// TwinCAT 3 PLC project PupunPLC
// ProgramVersion: 3.1.4024.0
// libraries:
//   Tc2_Standard, * (Beckhoff Automation GmbH)
//   Tc2_System, * (Beckhoff Automation GmbH)
//   Tc3_Module, * (Beckhoff Automation GmbH)
// project tree:
//   FactoryIO/GVLs/ GVL_Tutti.TcGVL
//   FactoryIO/TUTTITEHDAS/01 IN AND SORT/ FB_PICKNPLACE.TcPOU, FB_SPECIAL.TcPOU, FB_TURNTABLE.TcPOU, FB_WEIGHT.TcPOU
//   FactoryIO/TUTTITEHDAS/02 CNC/ FB_CNC_MILL.TcPOU, FB_WHEELSORT.TcPOU
//   FactoryIO/TUTTITEHDAS/03 BOXING/ FB_CLAMP.TcPOU, FB_SPECIAL_2.TcPOU, FB_TWO_AXIS_PICK.TcPOU
//   FactoryIO/TUTTITEHDAS/04 STORAGE/ FB_STACKER.TcPOU
//   FactoryIO/TUTTITEHDAS/CONVEYORS/ FB_CONVEYOR1.TcPOU
//   FactoryIO/TUTTITEHDAS/DUT/ S_NAMES_IN.TcDUT, S_NAMES_OUT.TcDUT, S_REGS_IN.TcDUT, S_REGS_OUT.TcDUT, U_TRANSLATE_IN.TcDUT, U_TRANSLATE_OUT.TcDUT, U_TRANSLATE_REGS_IN.TcDUT, U_TRANSLATE_REGS_OUT.TcDUT
//   FactoryIO/TUTTITEHDAS/ FBD_TUTTILINJASTO.TcPOU, MAIN_TUTTI.TcPOU, RUN.TcPOU
//   FactoryIO/TUTTITEHDAS/GVL/ TIO.TcGVL
//   GVLs/ GVL.TcGVL
//   / PlcTask.TcTTO
//   POUs/ MAIN.TcPOU
// real-time tasks:
//   TASK PlcTask: cycle T#10ms, priority 20, ADS port 350

CONFIGURATION PupunPLC
    RESOURCE PLC ON TwinCAT3
        TASK PlcTask(INTERVAL := T#10ms, PRIORITY := 20);
        PROGRAM MAIN WITH PlcTask : MAIN;
    END_RESOURCE
END_CONFIGURATION

// ---- FactoryIO/TUTTITEHDAS/DUT/S_NAMES_IN.TcDUT
TYPE S_NAMES_IN :
STRUCT
			
//===== 	BYTE	0		
iInput0		:		BIT;
iInput1		:		BIT;
iInput2		:		BIT;
iInput3		:		BIT;
iInput4		:		BIT;
iInput5		:		BIT;
iSensor6	:		BIT;
iInput7		:		BIT;
//===== 	BYTE	1	
iInput8		:		BIT;
iInput9		:		BIT;
iInput10	:		BIT;
iInput11	:		BIT;
iInput12	:		BIT;
iRetroSensor1	:		BIT;
iRetroSensor2	:		BIT;
iInput15	:		BIT;
//===== 	BYTE	2	
iSortLimit0	:		BIT;
iSortLimit90:		BIT;
iSortBackLimit	:		BIT;
iSortFrontLimit	:		BIT;
iPickPlace_Climit:		BIT;
iPickPlace_Z_Moving	:		BIT;
iPickPlace_XY_Moving	:		BIT;
iPickPlace_BoxDetected	:		BIT;
//===== 	BYTE	3	
iInput24	:		BIT;
iInput25	:		BIT;
iInput26	:		BIT;
iInput27	:		BIT;
iInput28	:		BIT;
iInput29	:		BIT;
iPusherBackLimit	:		BIT;
iPusherFrontLimit	:		BIT;
//===== 	BYTE	4	
iInput32	:		BIT;
iInput33	:		BIT;
iInput34	:		BIT;
iSensor5	:		BIT;
iInput36	:		BIT;
iInput37	:		BIT;
iInput38	:		BIT;
iInput39	:		BIT;
//===== 	BYTE	5	
iCNC1_Opened	:		BIT;
iCNC1_Busy	:		BIT;
iCNC1_Error	:		BIT;
iCNC2_Opened	:		BIT;
iCNC2_Busy	:		BIT;
iCNC2_Error	:		BIT;
iCNC3_Opened	:		BIT;
iCNC3_Busy	:		BIT;
//===== 	BYTE	6	
iCNC3_Error	:		BIT;
iInput49	:		BIT;
iInput50	:		BIT;
iInput51	:		BIT;
iInput52	:		BIT;
iInput53	:		BIT;
iTwoAxisPick1_ItemDetected	:		BIT;
iSensor10	:		BIT;
//===== 	BYTE	7	
iClamp1_Limit	:		BIT;
iClamp1_Clamped	:		BIT;
iInput58	:		BIT;
iInput59	:		BIT;
iInput60	:		BIT;
iInput61	:		BIT;
Sensor11	:		BIT;
Stacker1_LeftLimit	:		BIT;
//===== 	BYTE	8	
Stacker1_RightLimit	:		BIT;
Stacker1_MiddleLimit:		BIT;
iInput66	:		BIT;
iInput67	:		BIT;
iInput68	:		BIT;
iInput69	:		BIT;
iInput70	:		BIT;
iInput71	:		BIT;
//===== 	BYTE	9	
iInput72	:		BIT;
iInput73	:		BIT;
iInput74	:		BIT;
iInput75	:		BIT;
iInput76	:		BIT;
iInput77	:		BIT;
iInput78	:		BIT;
iInput79	:		BIT;
//===== 	BYTE	10	
iInput80	:		BIT;
iInput81	:		BIT;
iInput82	:		BIT;
iInput83	:		BIT;
iInput84	:		BIT;
iInput85	:		BIT;
iInput86	:		BIT;
iInput87	:		BIT;
//===== 	BYTE	11	
iInput88	:		BIT;
iInput89	:		BIT;
iInput90	:		BIT;
iInput91	:		BIT;
iInput92	:		BIT;
iInput93	:		BIT;
iInput94	:		BIT;
iInput95	:		BIT;
//===== 	BYTE	12	
iInput96	:		BIT;
iInput97	:		BIT;
iInput98	:		BIT;
iInput99	:		BIT;
iInput100	:		BIT;
iInput101	:		BIT;
iInput102	:		BIT;
iInput103	:		BIT;
//===== 	BYTE	13	
iInput104	:		BIT;
iInput105	:		BIT;
iInput106	:		BIT;
iInput107	:		BIT;
iInput108	:		BIT;
iInput109	:		BIT;
iInput110	:		BIT;
iInput111	:		BIT;
//===== 	BYTE	14	
iInput112	:		BIT;
iInput113	:		BIT;
iInput114	:		BIT;
iInput115	:		BIT;
iInput116	:		BIT;
iInput117	:		BIT;
iInput118	:		BIT;
iInput119	:		BIT;
//===== 	BYTE	15	
iInput120	:		BIT;
iInput121	:		BIT;
iInput122	:		BIT;
iInput123	:		BIT;
iInput124	:		BIT;
iInput125	:		BIT;
iInput126	:		BIT;
iInput127	:		BIT;
//===== 	BYTE	16	
iInput128	:		BIT;
iInput129	:		BIT;
iInput130	:		BIT;
iInput131	:		BIT;
iInput132	:		BIT;
iInput133	:		BIT;
iInput134	:		BIT;
iInput135	:		BIT;
//===== 	BYTE	17	
iInput136	:		BIT;
iInput137	:		BIT;
iInput138	:		BIT;
iInput139	:		BIT;
iInput140	:		BIT;
iInput141	:		BIT;
iInput142	:		BIT;
iInput143	:		BIT;
//===== 	BYTE	18	
iInput144	:		BIT;
iInput145	:		BIT;
iInput146	:		BIT;
iInput147	:		BIT;
iInput148	:		BIT;
iInput149	:		BIT;
iInput150	:		BIT;
iInput151	:		BIT;
//===== 	BYTE	19	
iInput152	:		BIT;
iInput153	:		BIT;
iInput154	:		BIT;
iInput155	:		BIT;
iInput156	:		BIT;
iInput157	:		BIT;
iInput158	:		BIT;
iInput159	:		BIT;
//===== 	BYTE	20	
iInput160	:		BIT;
iInput161	:		BIT;
iInput162	:		BIT;
iInput163	:		BIT;
iInput164	:		BIT;
iInput165	:		BIT;
iInput166	:		BIT;
iInput167	:		BIT;
//===== 	BYTE	21	
iInput168	:		BIT;
iInput169	:		BIT;
iInput170	:		BIT;
iInput171	:		BIT;
iInput172	:		BIT;
iInput173	:		BIT;
iInput174	:		BIT;
iInput175	:		BIT;
//===== 	BYTE	22	
iInput176	:		BIT;
iInput177	:		BIT;
iInput178	:		BIT;
iInput179	:		BIT;
iInput180	:		BIT;
iInput181	:		BIT;
iInput182	:		BIT;
iInput183	:		BIT;
//===== 	BYTE	23	
iInput184	:		BIT;
iInput185	:		BIT;
iInput186	:		BIT;
iInput187	:		BIT;
iInput188	:		BIT;
iInput189	:		BIT;
iInput190	:		BIT;
iInput191	:		BIT;
//===== 	BYTE	24	
iInput192	:		BIT;
iInput193	:		BIT;
iInput194	:		BIT;
iInput195	:		BIT;
iInput196	:		BIT;
iInput197	:		BIT;
iInput198	:		BIT;
iInput199	:		BIT;
//===== 	BYTE	25	
iInput200	:		BIT;
iInput201	:		BIT;
iInput202	:		BIT;
iInput203	:		BIT;
iInput204	:		BIT;
iInput205	:		BIT;
iInput206	:		BIT;
iInput207	:		BIT;
//===== 	BYTE	26	
iInput208	:		BIT;
iInput209	:		BIT;
iInput210	:		BIT;
iInput211	:		BIT;
iInput212	:		BIT;
iInput213	:		BIT;
iInput214	:		BIT;
iInput215	:		BIT;
//===== 	BYTE	27	
iInput216	:		BIT;
iInput217	:		BIT;
iInput218	:		BIT;
iInput219	:		BIT;
iInput220	:		BIT;
iInput221	:		BIT;
iInput222	:		BIT;
iInput223	:		BIT;
//===== 	BYTE	28	
iInput224	:		BIT;
iInput225	:		BIT;
iInput226	:		BIT;
iInput227	:		BIT;
iInput228	:		BIT;
iInput229	:		BIT;
iInput230	:		BIT;
iInput231	:		BIT;
//===== 	BYTE	29	
iInput232	:		BIT;
iInput233	:		BIT;
iInput234	:		BIT;
iInput235	:		BIT;
iInput236	:		BIT;
iInput237	:		BIT;
iInput238	:		BIT;
iInput239	:		BIT;
//===== 	BYTE	30	
iInput240	:		BIT;
iInput241	:		BIT;
iInput242	:		BIT;
iInput243	:		BIT;
iInput244	:		BIT;
iInput245	:		BIT;
iInput246	:		BIT;
iInput247	:		BIT;
//===== 	BYTE	31	
iInput248	:		BIT;
iInput249	:		BIT;
iInput250	:		BIT;
iInput251	:		BIT;
iInput252	:		BIT;
iInput253	:		BIT;
iInput254	:		BIT;
iInput255	:		BIT;
//===== 	BYTE	32	
iInput256	:		BIT;
iInput257	:		BIT;
iInput258	:		BIT;
iInput259	:		BIT;
iInput260	:		BIT;
iInput261	:		BIT;
iInput262	:		BIT;
iInput263	:		BIT;
//===== 	BYTE	33	

	
END_STRUCT
END_TYPE

// ---- FactoryIO/TUTTITEHDAS/DUT/S_NAMES_OUT.TcDUT
TYPE S_NAMES_OUT :
STRUCT
			
//===== 	BYTE	0	
//Kaheksan ekaa outputtia, GRANDES LUCES
oCoil0	:		BIT;
oCoil1	:		BIT;
oCoil2	:		BIT;
oCoil3	:		BIT;
oCoil4	:		BIT;
oCoil5	:		BIT;
oCoil6	:		BIT;
oCoil7	:		BIT;
//===== 	BYTE	1	
oEmitter1 :		BIT;
oEmitter2	:		BIT;
oRoller1	:		BIT;
oRoller2	:		BIT;
oRollerPick1	:	BIT;
oRollerSort1	:	BIT;
oRoller3	:		BIT;
oRemover2	:		BIT;
//===== 	BYTE	2	
oCoil16	:		BIT;
oCoil17	:		BIT;
oCoil18	:		BIT;
oCoil19	:		BIT;
oPickPlaceCplus	:		BIT;
oPickPlaceGrab	:		BIT;
oBelt1	:		BIT;
oBelt2	:		BIT;
//===== 	BYTE	3	
oBelt3	:		BIT;
oBelt4	:		BIT;
oBelt5	:		BIT;
oBelt6	:		BIT;
oScale1Plus	:			BIT;
oScale1Minus	:		BIT;
oPusher1	:			BIT;
oBelt7	:		BIT;
//===== 	BYTE	4	
oBelt8	:		BIT;
oStopBlade2	:		BIT;
oBelt9	:		BIT;
oWheelSort1Plus	:		BIT;
oWheelSort1Left	:		BIT;
oWheelSort1Right:		BIT;
oCoil38	:		BIT;
oCoil39	:		BIT;
//===== 	BYTE	5	
oCNC1_Start	:		BIT;
oCNC2_Start	:		BIT;
oCNC3_Start	:		BIT;
oCNC1_Lids	:		BIT;
oCNC2_Lids	:		BIT;
oCNC3_Lids	:		BIT;
oBelt12	:		BIT;
oBelt13	:		BIT;
//===== 	BYTE	6	
oBelt14	:		BIT;
oBelt15	:		BIT;
oRoller10	:		BIT;
oRoller11	:		BIT;
oRoller12	:		BIT;
oRoller13	:		BIT;
oStopBlade1	:		BIT;
oTwoAxisPick1_Grab	:		BIT;
//===== 	BYTE	7	
oRightPosit1_Clamp	:		BIT;
oRightPosit1_Raise	:		BIT;
oStackLight3_Red	:		BIT;
oStackLight3_Yellow	:		BIT;
oStackLight3_Green	:		BIT;
oEmitter4	:		BIT;
oCoil62	:			BIT;
Stacker1_Left	:	BIT;
//===== 	BYTE	8	
Stacker1_Right	:		BIT;
LoadingConveyor1:		BIT;
oCoil66	:		BIT;
oCoil67	:		BIT;
oCoil68	:		BIT;
oCoil69	:		BIT;
oCoil70	:		BIT;
oCoil71	:		BIT;
//===== 	BYTE	9	
oCoil72	:		BIT;
oCoil73	:		BIT;
oCoil74	:		BIT;
oCoil75	:		BIT;
oCoil76	:		BIT;
oCoil77	:		BIT;
oCoil78	:		BIT;
oCoil79	:		BIT;
//===== 	BYTE	10	
oCoil80	:		BIT;
oCoil81	:		BIT;
oCoil82	:		BIT;
oCoil83	:		BIT;
oCoil84	:		BIT;
oCoil85	:		BIT;
oCoil86	:		BIT;
oCoil87	:		BIT;
//===== 	BYTE	11	
oCoil88	:		BIT;
oCoil89	:		BIT;
oCoil90	:		BIT;
oCoil91	:		BIT;
oCoil92	:		BIT;
oCoil93	:		BIT;
oCoil94	:		BIT;
oCoil95	:		BIT;
//===== 	BYTE	12	
oCoil96	:		BIT;
oCoil97	:		BIT;
oCoil98	:		BIT;
oCoil99	:		BIT;
oCoil100	:		BIT;
oCoil101	:		BIT;
oCoil102	:		BIT;
oCoil103	:		BIT;
//===== 	BYTE	13	
oCoil104	:		BIT;
oCoil105	:		BIT;
oCoil106	:		BIT;
oCoil107	:		BIT;
oCoil108	:		BIT;
oCoil109	:		BIT;
oCoil110	:		BIT;
oCoil111	:		BIT;
//===== 	BYTE	14	
oCoil112	:		BIT;
oCoil113	:		BIT;
oCoil114	:		BIT;
oCoil115	:		BIT;
oCoil116	:		BIT;
oCoil117	:		BIT;
oCoil118	:		BIT;
oCoil119	:		BIT;
//===== 	BYTE	15	
oCoil120	:		BIT;
oCoil121	:		BIT;
oCoil122	:		BIT;
oCoil123	:		BIT;
oCoil124	:		BIT;
oCoil125	:		BIT;
oCoil126	:		BIT;
oCoil127	:		BIT;
//===== 	BYTE	16	
oCoil128	:		BIT;
oCoil129	:		BIT;
oCoil130	:		BIT;
oCoil131	:		BIT;
oCoil132	:		BIT;
oCoil133	:		BIT;
oCoil134	:		BIT;
oCoil135	:		BIT;
//===== 	BYTE	17	
oCoil136	:		BIT;
oCoil137	:		BIT;
oCoil138	:		BIT;
oCoil139	:		BIT;
oCoil140	:		BIT;
oCoil141	:		BIT;
oCoil142	:		BIT;
oCoil143	:		BIT;
//===== 	BYTE	18	
oCoil144	:		BIT;
oCoil145	:		BIT;
oCoil146	:		BIT;
oCoil147	:		BIT;
oCoil148	:		BIT;
oCoil149	:		BIT;
oCoil150	:		BIT;
oCoil151	:		BIT;
//===== 	BYTE	19	
oCoil152	:		BIT;
oCoil153	:		BIT;
oCoil154	:		BIT;
oCoil155	:		BIT;
oCoil156	:		BIT;
oCoil157	:		BIT;
oCoil158	:		BIT;
oCoil159	:		BIT;
//===== 	BYTE	20	
oCoil160	:		BIT;
oCoil161	:		BIT;
oCoil162	:		BIT;
oCoil163	:		BIT;
oCoil164	:		BIT;
oCoil165	:		BIT;
oCoil166	:		BIT;
oCoil167	:		BIT;
//===== 	BYTE	21	
oCoil168	:		BIT;
oCoil169	:		BIT;
oCoil170	:		BIT;
oCoil171	:		BIT;
oCoil172	:		BIT;
oCoil173	:		BIT;
oCoil174	:		BIT;
oCoil175	:		BIT;
//===== 	BYTE	22	
oCoil176	:		BIT;
oCoil177	:		BIT;
oCoil178	:		BIT;
oCoil179	:		BIT;
oCoil180	:		BIT;
oCoil181	:		BIT;
oCoil182	:		BIT;
oCoil183	:		BIT;
//===== 	BYTE	23	
oCoil184	:		BIT;
oCoil185	:		BIT;
oCoil186	:		BIT;
oCoil187	:		BIT;
oCoil188	:		BIT;
oCoil189	:		BIT;
oCoil190	:		BIT;
oCoil191	:		BIT;
//===== 	BYTE	24	
oCoil192	:		BIT;
oCoil193	:		BIT;
oCoil194	:		BIT;
oCoil195	:		BIT;
oCoil196	:		BIT;
oCoil197	:		BIT;
oCoil198	:		BIT;
oCoil199	:		BIT;
//===== 	BYTE	25	
oCoil200	:		BIT;
oCoil201	:		BIT;
oCoil202	:		BIT;
oCoil203	:		BIT;
oCoil204	:		BIT;
oCoil205	:		BIT;
oCoil206	:		BIT;
oCoil207	:		BIT;
//===== 	BYTE	26	
oCoil208	:		BIT;
oCoil209	:		BIT;
oCoil210	:		BIT;
oCoil211	:		BIT;
oCoil212	:		BIT;
oCoil213	:		BIT;
oCoil214	:		BIT;
oCoil215	:		BIT;
//===== 	BYTE	27	
oCoil216	:		BIT;
oCoil217	:		BIT;
oCoil218	:		BIT;
oCoil219	:		BIT;
oCoil220	:		BIT;
oCoil221	:		BIT;
oCoil222	:		BIT;
oCoil223	:		BIT;
//===== 	BYTE	28	
oCoil224	:		BIT;
oCoil225	:		BIT;
oCoil226	:		BIT;
oCoil227	:		BIT;
oCoil228	:		BIT;
oCoil229	:		BIT;
oCoil230	:		BIT;
oCoil231	:		BIT;
//===== 	BYTE	29	
oCoil232	:		BIT;
oCoil233	:		BIT;
oCoil234	:		BIT;
oCoil235	:		BIT;
oCoil236	:		BIT;
oCoil237	:		BIT;
oCoil238	:		BIT;
oCoil239	:		BIT;
//===== 	BYTE	30	
oCoil240	:		BIT;
oCoil241	:		BIT;
oCoil242	:		BIT;
oCoil243	:		BIT;
oCoil244	:		BIT;
oCoil245	:		BIT;
oCoil246	:		BIT;
oCoil247	:		BIT;
//===== 	BYTE	31	
oCoil248	:		BIT;
oCoil249	:		BIT;
oCoil250	:		BIT;
oCoil251	:		BIT;
oCoil252	:		BIT;
oCoil253	:		BIT;
oCoil254	:		BIT;
oCoil255	:		BIT;
//===== 	BYTE	32	
oCoil256	:		BIT;
oCoil257	:		BIT;
oCoil258	:		BIT;
oCoil259	:		BIT;
oCoil260	:		BIT;
oCoil261	:		BIT;
oCoil262	:		BIT;
oCoil263	:		BIT;
//===== 	BYTE	33	

END_STRUCT
END_TYPE

// ---- FactoryIO/TUTTITEHDAS/DUT/S_REGS_IN.TcDUT
TYPE S_REGS_IN :
STRUCT

//==== MEMORY REGISTERS IN				
nPickPlace1_X	:		WORD;	
nPickPlace1_Y	:		WORD;	
nPickPlace1_Z	:		WORD;	
nConveyorScaleWeight1 :	WORD;	
nRFID1_Status	:		WORD;	
nRFID1_ReadData	:		WORD;	
nRFID1_CommandID:		WORD;	
nTwoAxisPick1_X	:		WORD;	
nTwoAxisPick1_Z	:		WORD;	
nVisionSensor1_Value:	WORD;	
Stacker1_XPos	:		WORD;	
Stacker1_ZPos	:		WORD;	
nMemIn12	:		WORD;	
nMemIn13	:		WORD;	
nMemIn14	:		WORD;	
nMemIn15	:		WORD;	
nMemIn16	:		WORD;	
nMemIn17	:		WORD;	
nMemIn18	:		WORD;	
nMemIn19	:		WORD;	
nMemIn20	:		WORD;	
nMemIn21	:		WORD;	
nMemIn22	:		WORD;	
nMemIn23	:		WORD;	
nMemIn24	:		WORD;	
nMemIn25	:		WORD;	
nMemIn26	:		WORD;	
nMemIn27	:		WORD;	
nMemIn28	:		WORD;	
nMemIn29	:		WORD;	
nMemIn30	:		WORD;	
nMemIn31	:		WORD;	
nMemIn32	:		WORD;	



END_STRUCT
END_TYPE

// ---- FactoryIO/TUTTITEHDAS/DUT/S_REGS_OUT.TcDUT
TYPE S_REGS_OUT :
STRUCT
	
//==== MEMORY REGISTERS OUT			
nSetPickPlace1_X	:		WORD;
nSetPickPlace1_Y	:		WORD;
nSetPickPlace1_Z	:		WORD;
nRFID1_CodeAssign	:		WORD;
nRFID1_Command	:			WORD;
nRFID1_WriteData	:		WORD;
nRFID1_MemIndex	:			WORD;
nTwoAxisPick1_SetX	:		WORD;
nTwoAxisPick1_SetZ	:		WORD;
nDisplayPartCount	:		WORD;
nMemout10	:				WORD;
Disp_XCell	:				WORD;
Disp_ZCell	:				WORD;
Disp_XCellCoords	:		WORD;
Disp_ZCellCoords	:		WORD;
Stacker1_SETX	:		WORD;
Stacker1_SETZ	:		WORD;
nMemOut17	:		WORD;
nMemOut18	:		WORD;
nMemOut19	:		WORD;
nMemOut20	:		WORD;
nMemOut21	:		WORD;
nMemOut22	:		WORD;
nMemOut23	:		WORD;
nMemOut24	:		WORD;
nMemOut25	:		WORD;
nMemOut26	:		WORD;
nMemOut27	:		WORD;
nMemOut28	:		WORD;
nMemOut29	:		WORD;
nMemOut30	:		WORD;
nMemOut31	:		WORD;
nMemOut32	:		WORD;



END_STRUCT
END_TYPE

// ---- FactoryIO/TUTTITEHDAS/DUT/U_TRANSLATE_IN.TcDUT
TYPE U_TRANSLATE_IN :
UNION
	nArray :	ARRAY[0..15] OF BYTE;
	Label :		S_NAMES_IN;
END_UNION
END_TYPE

// ---- FactoryIO/TUTTITEHDAS/DUT/U_TRANSLATE_OUT.TcDUT
TYPE U_TRANSLATE_OUT :
UNION
	nArray :	ARRAY[0..15] OF BYTE;
	Label :		S_NAMES_OUT;
END_UNION
END_TYPE

// ---- FactoryIO/TUTTITEHDAS/DUT/U_TRANSLATE_REGS_IN.TcDUT
TYPE U_TRANSLATE_REGS_IN :
UNION
	nArray :	ARRAY [0..31] OF WORD;
	Label : 	S_REGS_IN;
END_UNION
END_TYPE

// ---- FactoryIO/TUTTITEHDAS/DUT/U_TRANSLATE_REGS_OUT.TcDUT
TYPE U_TRANSLATE_REGS_OUT :
UNION
	nArray :	ARRAY [0..31] OF WORD;
	Label :		S_REGS_OUT;
END_UNION
END_TYPE

// ---- FactoryIO/GVLs/GVL_Tutti.TcGVL
{attribute 'qualified_only'}
VAR_GLOBAL

END_VAR

VAR_GLOBAL PERSISTENT
	h : BOOL;
END_VAR

// ---- FactoryIO/TUTTITEHDAS/GVL/TIO.TcGVL
//{attribute 'qualified_only'}
VAR_GLOBAL
	//Factory IO
	FIN 	AT %I* 		: 	U_TRANSLATE_IN;  		//Inputit 0-15 Factory IO
	FOUT 	AT %Q*		: 	U_TRANSLATE_OUT;		//Outputit 0-15 Factory IO
	FMIN 	AT %MB0 	: 	U_TRANSLATE_REGS_IN; 	//Register In Factory IO
	FMOUT 	AT %MB64	: 	U_TRANSLATE_REGS_OUT;	//Register Out Factory IO

END_VAR

// ---- GVLs/GVL.TcGVL
{attribute 'qualified_only'}

VAR_GLOBAL
	
//	IO_Module_1 : IOModuleData;
//	IO_Temperature	AT %I*: 	TemperatureData;
{attribute 'OPC.UA.DA' := '3'}
	cIO_Out			AT %Q*:		ARRAY[1..4] OF BOOL;	
	cIO_In			AT %I*:		ARRAY[1..4] OF BOOL;	
	
	
// Link 'useless' variables to IO
	EthercatDevState 	AT%I*: UINT;
	Term2DevState 		AT%I*: UINT;
	EthercatDevCtrl 	AT%Q*: UINT;
	EthercatDev1		AT%I*: UINT;
	EthercatDev2		AT%I*: UINT;
	EthercatDev3		AT%I*: UINT;
END_VAR

// ---- POUs/MAIN.TcPOU
PROGRAM MAIN
VAR 
{attribute 'OPC.UA.DA' := '1'}
    hi:BOOL;
    timer: ton;
	{attribute 'OPC.UA.DA' := '1'}
	FIO_Input : BOOL;
{attribute 'OPC.UA.DA' := '1'}
	FIO_Output : BOOL; 
	testbit: BOOL;
END_VAR

// U; Pupu
// PW: 1

(*SUUNNITELMA
Vain pari structia missä on {attribute} päällä eli menee opc:lle jakoon
Niiden alle keräis jollain logiikalla kaikki jaettavat muuttujat.
	Simuloiden tilannetta missä asiakkaalle pitäisi se jakaa
	"tärkeät" asiat eli merkityksellinen data
	Toiminnallinen data
Laitekohtaisesti ryhmitelty? 
Erikseen vielä in/out ryhmä missä tietoa vois vaihtaa HMI:lle tms

PART 2
Toteutetaan hiukan OOP tai POP -tyyliä -> Vähennetään GVL käyttöä
Sagatowskin "PLC programming using TwinCAT 3 - Function blocks & interfaces (Part 6a/18)" video
	On käytössä valmista koodia mitä jokatapauksessa tulee muokattua niin voi heitellä ympäriinsä ja järjestellä mieluisaksi
	
*)

testbit := FIO_Output;

timer(IN := NOT timer.Q, PT := T#1S) ;
IF timer.Q THEN
    hi := NOT hi;
	FIO_Input := NOT FIO_Input;
END_IF

END_PROGRAM

// ---- FactoryIO/TUTTITEHDAS/01 IN AND SORT/FB_PICKNPLACE.TcPOU
FUNCTION_BLOCK FB_PICKNPLACE
VAR_INPUT
	IN :		BOOL;	//Power/Main switch
	Run : 		BOOL;	//Signal from previous state to start doing stuff
	Sensor1 :	BOOL;	//Diff sensor placed at the height of box
	MovingZ :	BOOL;
	MovingXY :	BOOL;
	BoxDetect :	BOOL;
	nPosX :	WORD;
	nPosY :	WORD;
	nPosZ :	WORD;
	
END_VAR
VAR_OUTPUT
	Q :			BOOL;
	Status: 	STRING;
	Go :		BOOL;
	
	Infeed :		BOOL;	//Conveyor
	Outfeed :		BOOL;	//Conveyor
	Grab :		BOOL;
	CPlus :		BOOL;
	RegSetX :		WORD;
	RegSetY : 		WORD;
	RegSetZ :		WORD;	
	
END_VAR
VAR
	iState: INT;
	fbTON : 	TON;
	
END_VAR


IF NOT IN THEN
	Q := FALSE;
	iState := 0;
	ELSE
		Q := TRUE;
END_IF

CASE iState OF
	
0: //idle
	Status := 		'0 - Idle';
	IF Q THEN
		iState := 10;
	END_IF
10: //feed in
	Status := 		'10 - Feed in';
	Go :=			FALSE;
	IF Run THEN
		Infeed := 	TRUE;
		iState := 	20;
	END_IF
20: //Align and stop
	Status := 		'20 - Box in place, go fetch';
	IF Sensor1 THEN
		Infeed :=	FALSE;
		RegSetX :=	850;
		RegSetY :=	660;
		RegSetZ :=	0; 	//1000;
		iState := 	21;
	END_IF
21: //Go down
	Status := 		'21 - Above the box, go pick it';
	IF nPosX > 700 THEN
		RegSetZ :=	1000;
		iState := 	30;
	END_IF
30: //Grab it and go
	Status := 		'30 - Box detected, grabbing';
	IF BoxDetect THEN
		Grab :=		TRUE;
		//hold for little while
		fbTON(IN := TRUE, PT := T#200MS);
		IF fbTON.Q THEN
			fbTON(IN := FALSE);
			RegSetX :=	0;		//Over the outfeed conveyor
			RegSetY :=	530;
			RegSetZ :=	280;
			Go :=		TRUE;
			iState := 	40; 
		END_IF
	END_IF
40: //Roll out
	Status := 		'40 - Roll out';
	IF NOT MovingXY AND NOT Sensor1 THEN
 	Grab := 	FALSE;
	Infeed := 	TRUE;
	Outfeed :=	TRUE;
	iState := 	10;
	END_IF
END_CASE

END_FUNCTION_BLOCK

// ---- FactoryIO/TUTTITEHDAS/RUN.TcPOU
FUNCTION_BLOCK RUN
VAR_INPUT
	IN:		BOOL;
	
END_VAR
VAR_OUTPUT
	Q :		 BOOL;
	PWR_LIGHT1 :BOOL;
	Emitter1 :	BOOL;
	LIGHT0:		BOOL;
	LIGHT1:		BOOL;
	LIGHT2:		BOOL;
	LIGHT3:		BOOL;
	LIGHT4:		BOOL;
	LIGHT5:		BOOL;
	LIGHT6:		BOOL;
	LIGHT7:		BOOL;
	
END_VAR
VAR
	iState: 	INT;
	fbTON : 	TON;
	WaitTime :	TIME := T#1000MS;
	iNextState: INT;
	iStateHeartBeat: INT;
	Run_It: BOOL;
END_VAR

//home-made R_TRIG. No stop-button yet though
IF IN = TRUE AND Run_It = FALSE THEN
	Run_It := IN;
END_IF

IF Run_It THEN
	PWR_LIGHT1 := 	TRUE;
	Q := 			TRUE;
	Emitter1 :=		TRUE;
END_IF


CASE iState OF
		0: //IDLE
			LIGHT0 := FALSE;
			LIGHT1 := FALSE;
			LIGHT2 := FALSE;
			LIGHT3 := FALSE;
			LIGHT4 := FALSE;
			LIGHT5 := FALSE;
			LIGHT6 := FALSE;
			LIGHT7 := FALSE;
			iStateHeartBeat := iStateHeartBeat+1;
			IF Q THEN 
				iState := 10;
			END_IF
		10:	
			fbTON(IN:= TRUE, PT:= WaitTime);
			IF fbTON.Q THEN
				fbTON(IN := FALSE);
				LIGHT1 := TRUE;
				LIGHT0 := FALSE;
				iState := iState+1;
				iStateHeartBeat := iStateHeartBeat+1;
			END_IF
		11:
			fbTON(IN:= TRUE, PT:= WaitTime);
			IF fbTON.Q THEN
				fbTON(IN := FALSE);
				LIGHT2 := TRUE;
				LIGHT1 := FALSE;
				iState := iState+1;
				iStateHeartBeat := iStateHeartBeat+1;
			END_IF
		12:
			fbTON(IN:= TRUE, PT:= WaitTime);
			IF fbTON.Q THEN
				fbTON(IN := FALSE);
				LIGHT3 := TRUE;
				LIGHT2 := FALSE;
				iState := iState+1;
				iStateHeartBeat := iStateHeartBeat+1;
			END_IF
		13:
			fbTON(IN:= TRUE, PT:= WaitTime);
			IF fbTON.Q THEN
				fbTON(IN := FALSE);
				LIGHT4 := TRUE;
				LIGHT3 := FALSE;
				iState := iState+1;
				iStateHeartBeat := iStateHeartBeat+1;
			END_IF
		14:
			fbTON(IN:= TRUE, PT:= WaitTime);
			IF fbTON.Q THEN
				fbTON(IN := FALSE);
				LIGHT5 := TRUE;
				LIGHT4 := FALSE;
				iState := iState+1;
				iStateHeartBeat := iStateHeartBeat+1;
			END_IF
		15:
			fbTON(IN:= TRUE, PT:= WaitTime);
			IF fbTON.Q THEN
				fbTON(IN := FALSE);
				LIGHT6 := TRUE;
				LIGHT5 := FALSE;
				iState := iState+1;
				iStateHeartBeat := iStateHeartBeat+1;
			END_IF
		16:
			fbTON(IN:= TRUE, PT:= WaitTime);
			IF fbTON.Q THEN
				fbTON(IN := FALSE);
				LIGHT7 := TRUE;
				LIGHT6 := FALSE;
				iState := iState+1;
				iStateHeartBeat := iStateHeartBeat+1;
			END_IF
		17:
			fbTON(IN:= TRUE, PT:= WaitTime);
			IF fbTON.Q THEN
				fbTON(IN := FALSE);
				LIGHT0 := TRUE;
				LIGHT7 := FALSE;
				iState := 10;
				iStateHeartBeat := iStateHeartBeat+1;
			END_IF
		END_CASE


//Ei toiminu, yritin ARRAYlla ja BYTEllä kontrolloida FOR i tyylillä valoja mutta parempi luovuttaa tältä erää
//		fbTON(IN:= TRUE, PT:= WaitTime);
//		IF fbTON.Q THEN
//		fbTON(IN := FALSE);
//			fbTON2(IN := TRUE, PT := WaitLights);

//			IF fbTON2.Q THEN
//				byLIGHT.i := TRUE;
//				//aLight[i-1] := FALSE;		//kokeillaas hiukan myöhemmin
//				i := i+1;
//				IF i > 7 THEN
//					i := 0;
//				END_IF
//				fbTON2(IN := FALSE);
//			END_IF
//		END_IF

END_FUNCTION_BLOCK

// ---- FactoryIO/TUTTITEHDAS/01 IN AND SORT/FB_SPECIAL.TcPOU
FUNCTION_BLOCK FB_SPECIAL
VAR_INPUT
	IN : 	BOOL;
	Run :	BOOL;		//Emitter = Run
	SpawnAmount : INT := 1;
//	Sensor : BOOL;		//mieluummin käytän ei sensoriin liittyvän ratkaisun
END_VAR
VAR_OUTPUT
	Q :			BOOL;
	Emitter : 	BOOL;	//Emitter = Run
	Remover :	BOOL;	//Remover = Run
END_VAR
VAR
	iState: INT;
	fbTON: TON;
	fbTON2: TON;
	X0: BOOL;
	i: INT;
END_VAR

IF NOT IN THEN
	Q := FALSE;
	iState := 0;
	ELSE
		Q := TRUE;
	//	Emitter := Run;		//Toimi ihan hyvin kun 1 kpl riittää
		Remover := Run;		
END_IF

IF Run = TRUE AND X0 = FALSE THEN
	X0 := TRUE;
END_IF

//äh, for-loopin tein ja se varmaan toimiki mutta aivan muualla oli bugi
IF X0 AND i < SpawnAmount THEN			//X sekunnin välein väläyttää Emitteriä SpawnAmountin verran (3 oletus)
	fbTON(IN := TRUE, PT := T#3000MS);
	IF fbTON.Q THEN
		Emitter := TRUE;
		fbTON2(IN:=TRUE, PT := T#100MS);
		IF fbTON2.Q THEN
			Emitter := FALSE;
			fbTON2(IN := FALSE);
			fbTON(IN := FALSE);
			i := i+1;
		END_IF
	END_IF
ELSE 
	X0 := 		FALSE;
	Emitter := 	FALSE;
	i := 		0;
END_IF

END_FUNCTION_BLOCK

// ---- FactoryIO/TUTTITEHDAS/01 IN AND SORT/FB_TURNTABLE.TcPOU
FUNCTION_BLOCK FB_TURNTABLE
VAR_INPUT
	IN :		BOOL;
	Limit90 :		BOOL;
	Limit0 :		BOOL;
	BackLimit :		BOOL;
	FrontLimit :	BOOL;
	
END_VAR
VAR_OUTPUT
	Q :		BOOL;
	Go :	BOOL;
	Status : 	STRING;
	RollPlus :	BOOL;
	RollMinus :	BOOL;
	Turn :		BOOL;

	
	//Feeding rollers
	FeedIn1 : BOOL;
	FeedOut1 : BOOL;
	FeedOut2 : BOOL;
END_VAR
VAR
	iState: INT;
	fbTON : TON;	
	
	fbTON2: TON;
END_VAR


IF NOT IN THEN
	Q := FALSE;
	iState := 0;
	ELSE
		Q := TRUE;
END_IF

CASE iState OF
	
0: //idle
	Status := 		'0 - Idle';
	RollPlus := 	FALSE;
	RollMinus := 	FALSE;
	Turn :=			FALSE;
	FeedIn1 :=		FALSE;
	IF Q THEN 
	iState := 10;	
	END_IF
	
10: //receive
	Status := 		'10 - Receive';
	FeedIn1 := 	TRUE;
	RollPlus := TRUE;
	IF FrontLimit THEN
		iState := 20;
	END_IF
	
20: //stop and turn
	Status := 		'20 - Turn';
	FeedIn1 :=	FALSE;
	RollPlus := FALSE;
	Turn := 	TRUE;
	IF Limit90 THEN
		iState := 	30;
	END_IF
	
30: //feed out
	Status := 		'30 - Feed out and wait 1s';
	RollMinus := 	TRUE;
	Go := 			TRUE;
	fbTON2(IN := TRUE, PT := T#1000MS);
	IF fbTON2.Q THEN fbTON2(IN := FALSE);
		IF NOT BackLimit THEN
		fbTON(IN := TRUE, PT := T#1000MS);
			IF fbTON.Q THEN	fbTON(IN := FALSE);
				Turn := 	FALSE;
				RollMinus := FALSE;
				iState := 	40;
			END_IF
		END_IF
	END_IF
	
40: //going back to start
	Status := 		'40 - Back to start';
	Go := 			FALSE;
	IF Limit0 THEN
		iState := 10;
	END_IF

END_CASE

END_FUNCTION_BLOCK

// ---- FactoryIO/TUTTITEHDAS/01 IN AND SORT/FB_WEIGHT.TcPOU
FUNCTION_BLOCK FB_WEIGHT
VAR_INPUT
	IN :	BOOL;
	Run :	BOOL;
	nWeight :		WORD;
	nSetWeightA : 	WORD := 400;
	nSetWeightB : 	WORD := 600;
	PusherFrontLimit : 	BOOL;
	PusherBackLimit :	BOOL;
	
END_VAR
VAR_OUTPUT
	Q :		BOOL;
	Status : INT;
	Go :	BOOL;		//Pusher etc. that reacts to weight
	ConveyorPlus : 	BOOL;
	ConveyorMinus :	BOOL;
	StopBlade :		BOOL;
	Pusher :		BOOL;
END_VAR
VAR
	iState: INT;
	fbTON: TON;
	fbTON2: TON;
END_VAR

IF NOT IN THEN
	Q := FALSE;
	iState := 0;
	ELSE
		Q := TRUE;
END_IF

Status := iState;

CASE iState OF
	0 : //Idle
	IF NOT Q THEN
	ConveyorPlus := 	FALSE;
	StopBlade :=		FALSE;
	ELSE
		iState :=			10;
	END_IF
	
	10 : //Feeding in
	ConveyorPlus := 	TRUE;
	Pusher := 			FALSE;
	IF nWeight > 100 THEN
		StopBlade :=		TRUE;
		fbTON(IN := TRUE, PT := T#1500MS);
		IF fbTON.Q THEN fbTON(IN := FALSE);
			ConveyorPlus :=		FALSE;
			iState :=			20;
		END_IF		
	END_IF
	
	20 : //JUDGING THE SINNERS ACCORDING TO THEIR WEIGHT
	fbTON2(IN := TRUE, PT := T#100MS);
	IF fbTON2.Q THEN fbTON2(IN := FALSE);
		IF nWeight > nSetWeightA AND nWeight < nSetWeightB THEN
			Pusher := 	TRUE;
			Go :=		TRUE;
			iState := 	30;
		END_IF
	END_IF
	
	30 : 
	fbTON2(IN := TRUE, PT := T#100MS);
	IF fbTON2.Q THEN fbTON2(IN := FALSE);
		Go :=		FALSE;
		IF PusherFrontLimit THEN
		Pusher := 	FALSE;
		StopBlade := FALSE;
		iState :=	40;
		END_IF
	END_IF

	40 :	//waiting for scale to clear
	IF PusherBackLimit THEN
		iState := 10;
	END_IF
END_CASE

END_FUNCTION_BLOCK

// ---- FactoryIO/TUTTITEHDAS/02 CNC/FB_CNC_MILL.TcPOU
FUNCTION_BLOCK FB_CNC_MILL
VAR_INPUT
	IN : BOOL;
	Opened	: BOOL;
	Busy	: BOOL;
	Error	: BOOL;
	mProgress : WORD;
END_VAR
VAR_OUTPUT
	Q		: BOOL;
	Start	: BOOL;
	Stop	: BOOL;
	Reset	: BOOL;
	Produce_Lids_Or_Dont	: BOOL;
END_VAR
VAR
	iState: INT;
END_VAR

IF NOT IN THEN
	Q := 		FALSE;
	Start := 	FALSE;
	ELSE
		Q := 		TRUE;
		Start := 	TRUE;
END_IF

END_FUNCTION_BLOCK

// ---- FactoryIO/TUTTITEHDAS/02 CNC/FB_WHEELSORT.TcPOU
FUNCTION_BLOCK FB_WHEELSORT
VAR_INPUT
	IN : 	BOOL;
	Sensor : BOOL;
END_VAR
VAR_OUTPUT
	Q :			BOOL;
	Plus :	BOOL;
	Left :	BOOL;
	Right :	BOOL;
END_VAR
VAR
	iState: INT;
	rTRIG : R_TRIG;
END_VAR

IF NOT IN THEN
	Q := FALSE;
	iState := 0;
	ELSE
		Q := 	TRUE;
		Plus := TRUE;
END_IF

//Nyt vain latoo yksi kerrallaan linjoille
//Myöhemmän ajan puuha tutkia jonotilanne ja sen mukaan päättää

CASE iState OF
0 : //Suoraan
	Left := 	FALSE;
	Right := 	FALSE;	

	rTRIG(CLK := Sensor);
	IF rTRIG.Q THEN
		iState := 1;
	END_IF
1 : //Vasen
	Left := 	TRUE;
	Right := 	FALSE;

	rTRIG(CLK:=Sensor);
	IF rTRIG.Q THEN
		iState := 2;
	END_IF
2 : //Oikea
	Left := 	FALSE;
	Right := 	TRUE;
		
	rTRIG(CLK:=Sensor);
	IF rTRIG.Q THEN
		iState := 0;
	END_IF
	
END_CASE

END_FUNCTION_BLOCK

// ---- FactoryIO/TUTTITEHDAS/03 BOXING/FB_CLAMP.TcPOU
FUNCTION_BLOCK FB_CLAMP
VAR_INPUT
	IN :	BOOL;
	Clamped :	BOOL;
	LimitUpDown :	BOOL;
	VisiSensor :	WORD;
	AllClear :			BOOL; 	//"All clear" -message from picker
END_VAR
VAR_OUTPUT
	Q : 		BOOL;
	StopBlade :	BOOL;
	Clamp :		BOOL;
	Raise :		BOOL;
	ReadyForPickUp: BOOL;
END_VAR
VAR
	iState: INT;
	fbTON: TON;
END_VAR

IF NOT IN THEN
	Q := FALSE;
	iState := 0;
	ELSE
		Q := TRUE;	
END_IF

CASE iState OF
	0 : //idle
	IF Q THEN
		iState := 10;
	END_IF
	10 : //wait for something to CLAMP
	IF VisiSensor = 0 THEN
		StopBlade := FALSE;
		ReadyForPickUp := FALSE;
		ELSE
			StopBlade := TRUE;
			iState := 20;
	END_IF
	20 : //CLAMP CLAMP CLAMP!
	fbTON(IN := TRUE, PT := T#500MS);
	IF fbTON.Q THEN fbTON(IN := FALSE);
		Clamp := TRUE;
		iState := 30;
	END_IF
	30 : //UNCLAMP
	IF Clamped THEN
		Clamp := FALSE;
		iState := 40;
		ReadyForPickUp := TRUE;
	END_IF
	40 : //Wait for all clear
	fbTON(IN := TRUE, PT := T#300MS);
	IF AllClear AND fbTON.Q THEN fbTON(IN := FALSE);
			StopBlade := FALSE;
			iState := 10;
	END_IF
	
END_CASE

END_FUNCTION_BLOCK

// ---- FactoryIO/TUTTITEHDAS/03 BOXING/FB_SPECIAL_2.TcPOU
FUNCTION_BLOCK FB_SPECIAL_2
VAR_INPUT
	IN : 	BOOL;
	Run :	BOOL;		//Emitter = Run
	SpawnAmount : INT := 2;
//	Sensor : BOOL;		//mieluummin käytän ei sensoriin liittyvän ratkaisun
END_VAR
VAR_OUTPUT
	Q :			BOOL;
	Emitter : 	BOOL;	//Emitter = Run
	Remover :	BOOL;	//Remover = Run
END_VAR
VAR
	iState: INT;
	fbTON: TON;
	fbTON2: TON;
	X0: BOOL;
	i: INT;
END_VAR

IF NOT IN THEN
	Q := FALSE;
	iState := 0;
	ELSE
		Q := TRUE;
	//	Emitter := Run;		//Toimi ihan hyvin kun 1 kpl riittää
		Remover := Run;		
END_IF

IF Run = TRUE AND X0 = FALSE THEN
	X0 := TRUE;
END_IF

//äh, for-loopin tein ja se varmaan toimiki mutta aivan muualla oli bugi
//kuten myös R_TRIGulla olis kannattanu... meni jo
IF X0 AND i < SpawnAmount THEN			//1s välein väläyttää Emitteriä SpawnAmountin verran (3 oletus)
	fbTON(IN := TRUE, PT := T#2000MS);
	IF fbTON.Q THEN
		Emitter := TRUE;
		fbTON2(IN:=TRUE, PT := T#100MS);
		IF fbTON2.Q THEN
			Emitter := FALSE;
			fbTON2(IN := FALSE);
			fbTON(IN := FALSE);
			i := i+1;
		END_IF
	END_IF
ELSE 
	X0 := 		FALSE;
	Emitter := 	FALSE;
	i := 		0;
END_IF

END_FUNCTION_BLOCK

// ---- FactoryIO/TUTTITEHDAS/03 BOXING/FB_TWO_AXIS_PICK.TcPOU
FUNCTION_BLOCK FB_TWO_AXIS_PICK
VAR_INPUT
	IN :	BOOL;
	PartReadyForPickup :	BOOL;	//Signal from other device
	PalletReady :	BOOL;			//Capacitive sensor looking for pallet in place
	PartDetected :	BOOL;			//Grabber sensor when part is near
	X_Position :	WORD;
	Z_Position :	WORD;
	
END_VAR
VAR_OUTPUT
	Q :			BOOL;
	AllClear :	BOOL;
	Busy :		BOOL;
	SetX :		WORD;
	SetZ :		WORD;
	Grab :		BOOL;
	PartCount :		WORD;
	Roller :	BOOL;

	
END_VAR
VAR
	iState: INT;
	fbTON: TON;
END_VAR

IF NOT IN THEN
	Q := FALSE;
	iState := 0;
	ELSE
		Q := TRUE;	
END_IF

CASE iState OF
	0 : //idle
	IF Q THEN
		iState := 10;
	END_IF
	10 : //waiting for stuff
		AllClear := TRUE;
		Busy := FALSE;
		SetX := 1000;
		SetZ := 200;

		IF NOT PalletReady THEN
		Roller :=	TRUE;
		ELSE
			Roller := FALSE;
		END_IF
		IF PartReadyForPickup THEN
			AllClear := FALSE;
		END_IF
		IF PartReadyForPickup AND PalletReady AND X_Position > 700 THEN
			iState := 11;
		END_IF
	11 :
		IF PartReadyForPickup THEN
		Busy := 	TRUE;
		AllClear := FALSE;
		SetZ := 1000;
		iState := 20;
		END_IF
	20 : //pick
		IF PartDetected THEN
		Grab := TRUE;
		iState := 30;
		END_IF
	30 : //Raise
		SetZ := 200;
		iState := 40;
	
	40 : 
		IF Z_Position < 300 THEN
		SetX := 110;
		iState := 50;
		END_IF
	50 : 
		IF X_Position < 300 THEN
		SetZ := 700;
		iState := 60;
		END_IF
	60 :
		IF Z_Position >650 THEN
		Grab := FALSE;
		fbTON(IN := TRUE, PT := T#200MS);
			IF fbTON.Q THEN fbTON(IN := FALSE);
			SetZ := 200;
			iState := 70;
			END_IF
		END_IF
	70 : 
		IF Z_Position < 500 THEN
		AllClear := TRUE;
		iState := 	80;
		END_IF
	80 :
		Roller := TRUE;
		IF NOT PalletReady THEN
		iState := 10;
		END_IF
	
END_CASE

END_FUNCTION_BLOCK

// ---- FactoryIO/TUTTITEHDAS/04 STORAGE/FB_STACKER.TcPOU
FUNCTION_BLOCK FB_STACKER
VAR_INPUT
	IN : 	BOOL;
	X_NextPalletGoesTo : INT := 1;	//Desired X-cell coordinate for next pallet
	Z_NextPalletGoesTo : INT := 1; 	//Desired Z-cell coordinate for next pallet
	Raise : BOOL;
	X_Position : WORD;	//Current pos reported from stacker
	Z_Position : WORD;	//Current pos reported from stacker
	Sensor :	BOOL;
	LeftLimit : BOOL;
	RightLimit : BOOL;
	MiddleLimit : 	BOOL;
	
END_VAR
VAR_OUTPUT
	Q : 	BOOL;
	Status: STRING;
	Busy : BOOL; 	//Signal that all clear when not true
	Set_X :	WORD;	//output coords to stacker
	Set_Z : WORD;	//output coords to stacker
	Left : 	BOOL;			//For loading/unloading pallet into device
	Right :	BOOL;			//For loading/unloading pallet into device
	Infeed : BOOL;			//Loading conveyor
	
	//Display stuff
		Display_X: WORD;	//Convenience display of coordinates
		Display_Z: WORD;	//Convenience display of coordinates
		Display_XCell : WORD;	//Convenience display of calculated cell
		Display_ZCell : WORD;	//Convenience display of calculated cell
	
END_VAR
VAR
	XCell : INT;	//X Cell number. Calculate coords from this
	ZCell : INT;	//Z Cell number. Calculate coords from this
	//Variables
		XSpace : INT	:= 107;		//104 Spacing in X-direction
		XOffset: INT	:= 144;		//offset //150;
		
		ZSpace : INT	:= 170;		//170
		ZOffset: INT	:= 30;		//30 
		Raise_Amount: 	INT;	//Changes in response to Raise:BOOL
		Raise_Amount_Variable : INT := 50;

	iState: INT;
	Raise_Wait :	TIME := T#1000MS;
	LoadWaiting: BOOL;
	fbTON: TON;

	X_NextPalletGoesTo_Var: INT := 1;
	Z_NextPalletGoesTo_Var: INT := 1;
END_VAR

IF NOT IN THEN
	Q := FALSE;
	iState := 0;
	ELSE
		Q := TRUE;	
END_IF

//To Actions or Methods?
//=======================================
	
	Display_X := Set_X;
	Display_Z := Set_Z;
	Display_XCell := TO_WORD(XCell);
	Display_ZCell := TO_WORD(ZCell);

//CALCULATIONS. Goes to start pos when coordinates are out of bound. Otherwise converts XCell to set-X coordinates for stacker machinen
	IF XCell = 0 THEN
		Set_X := TO_WORD(0);
		ELSE
		IF XCell >= 10 OR XCell < 0 THEN
			XCell := 0;
			ELSE
			Set_X := TO_WORD((XCell-1)*XSpace+XOffset);
		END_IF
	END_IF
	
	IF ZCell = 0 THEN
		Set_Z := TO_WORD(0+Raise_Amount);
		ELSE
			IF ZCell >= 7 OR ZCell < 0 THEN
				ZCell := 0;
				ELSE
				Set_Z := TO_WORD(
				((ZCell-1) *ZSpace) +ZOffset +Raise_Amount
				); 
			END_IF
	END_IF
	
//Raise = 50 higher when true. Variable in ZCell calculations
	IF NOT Raise THEN
		Raise_Amount := 0;
		ELSE
			Raise_Amount := Raise_Amount_Variable;
	END_IF

//Feed in
	IF NOT Sensor THEN
		Infeed := 		TRUE;
	//	LoadWaiting := 	FALSE;
		ELSE
			Infeed := 		FALSE;
			LoadWaiting := 	TRUE;
	END_IF

//=============================================

	
CASE iState OF
0 : //Idle
	Status := '0 - Idle. Waiting for power';
	IF Q THEN
		iState := 10;
		FeikkiHyllyttaja();
	END_IF
10 : //Start pos, Busy off if everything in 0, feed in
	Status := '10 - Start pos. All to home positions';
	IF X_Position = 0 AND Z_Position = 0 AND MiddleLimit THEN
	Busy := 	FALSE;
	iState := 	20;
	ELSE
		Busy := 	TRUE;
	END_IF

	IF NOT MiddleLimit THEN		//tarkoitus olisi tuoda kelkka sisään, sitten vasta liikkua
		Left := 	FALSE;
		Right :=	FALSE;
	ELSE 
		XCell := 	0;
		ZCell := 	0;
	END_IF
	
20 : //Load arrived, if all ok then proceed. Busy on
	Status := '20 - Waiting on pallet AND storage cell coordinates';
	IF LoadWaiting AND X_NextPalletGoesTO >= 1 THEN	
		Left := 	TRUE;
		iState := 	30;
		Busy :=		TRUE;
	END_IF
30 : //Action time. Raise load
	Status := '30 - Pallet arrived. Picking up';
	IF LeftLimit THEN
		Raise := 	TRUE;
		fbTON(IN := TRUE, PT := Raise_Wait);
		IF fbTON.Q THEN		fbTON(IN := FALSE);
			Left :=			FALSE;
			LoadWaiting := 	FALSE;
			iState := 		40;
		END_IF
	END_IF
40 : //Skiddledoo to right cell
	Status := '40 - Skiddledoo to correct cell coordinates';
	IF MiddleLimit THEN
		XCell := X_NextPalletGoesTo;	
		ZCell := Z_NextPalletGoesTo;	//pitää voida myös nollata nämä kun lava viety
		iState := 50;
	END_IF
50 : //Feed out load
	Status := '50 - Feeding pallet to storage';
	IF X_Position >= (Set_X-20) AND Z_Position >= (Set_Z-20) THEN
		X_NextPalletGoesTo := 0;
		Z_NextPalletGoesTo := 0;
		Right := 	TRUE;
		iState := 	60;
	END_IF
60 : //Skaddledoo back to start
	Status := '60 - Lower and retract';
	IF RightLimit THEN
		Raise := 	FALSE;
		fbTON(IN := TRUE, PT := Raise_Wait);
	END_IF
	
	IF fbTON.Q THEN 	fbTON(IN := FALSE);
		Right := 	FALSE;
		iState := 	70;
	END_IF
70 : //
	Status := '70 - Skaddledoo back to home pos';
	IF MiddleLimit THEN
			iState := 	0;
	END_IF

END_CASE

ACTION FeikkiHyllyttaja:

//IF X_NextPalletGoesTo_var >= 10 THEN
//	X_NextPalletGoesTo_Var := 1;
//	Z_NextPalletGoesTo_var := Z_NextPalletGoesTo_var+1;
//END_IF

//IF Z_NextPalletGoesTo_var >= 7 THEN
//	Z_NextPalletGoesTo_var := 1;
//END_IF

IF X_NextPalletGoesTo <= 0 THEN
		X_NextPalletGoesTo_var := 	X_NextPalletGoesTo_var+1;
	IF X_NextPalletGoesTo_var >= 10 OR X_NextPalletGoesTo_var <= 0 THEN
		X_NextPalletGoesTo_Var := 1;
		Z_NextPalletGoesTo_var := Z_NextPalletGoesTo_var+1;
	IF Z_NextPalletGoesTo_var >= 7 THEN
			Z_NextPalletGoesTo_var := 1;
	END_IF
	END_IF
END_IF
		X_NextPalletGoesTo := 		X_NextPalletGoesTo_var;
		Z_NextPalletGoesTo := 		Z_NextPalletGoesTo_var;
END_ACTION

END_FUNCTION_BLOCK

// ---- FactoryIO/TUTTITEHDAS/CONVEYORS/FB_CONVEYOR1.TcPOU
FUNCTION_BLOCK FB_CONVEYOR1
VAR_INPUT
	IN :		BOOL;	//When IN, then rollers and Q on
END_VAR
VAR_OUTPUT
	Q :		BOOL;
	ROLL1 :	BOOL;
	ROLL2 :	BOOL;
	ROLL3 :	BOOL;
	ROLL4 :	BOOL;
	ROLL5 :	BOOL;
	ROLL6 :	BOOL;
END_VAR
VAR
END_VAR

IF NOT IN THEN
	Q := FALSE;
	ROLL1 := FALSE;
	ROLL2 := FALSE;
	ROLL3 := FALSE;
	ROLL4 := FALSE;
	ROLL5 := FALSE;
	ROLL6 := FALSE;
	ELSE
		Q := 		TRUE;
		ROLL1 := 	TRUE;
		ROLL2 := 	TRUE;
		ROLL3 := 	TRUE;
		ROLL4 := 	TRUE;
		ROLL5 := 	TRUE;
		ROLL6 := 	TRUE;
END_IF

END_FUNCTION_BLOCK

// ---- FactoryIO/TUTTITEHDAS/FBD_TUTTILINJASTO.TcPOU
PROGRAM FBD_TUTTILINJASTO
VAR
	fbRUN: RUN;
	START_TO_SORT1: FB_CONVEYOR1;
	fbSORT1: FB_TURNTABLE;
	SORT_TO_PICKNPLACE: FB_CONVEYOR1;
	fbPICKNPLACE_1: FB_PICKNPLACE;
	fbSortByWeight: FB_WEIGHT;
	WEIGHT_TO_CNC: FB_CONVEYOR1;
	WEIGHT_TO_LIQUIDS: FB_CONVEYOR1;
	
	fbSpecial1: FB_SPECIAL;
	fbSpecial2: FB_SPECIAL_2;
	SORT_TO_CNC: FB_CONVEYOR1;
	fbWheelSort1: FB_WHEELSORT;
	fbCNCMill1: FB_CNC_MILL;
	fbCNCMill2: FB_CNC_MILL;
	fbCNCMill3: FB_CNC_MILL;
	CNC_TO_BOXING: FB_CONVEYOR1;
	BOXING_TO_STORAGE: FB_CONVEYOR1;
	fbClamp: FB_CLAMP;
	fbTwoAxisPick1: FB_TWO_AXIS_PICK;
	fbStacker1: FB_STACKER;
END_VAR

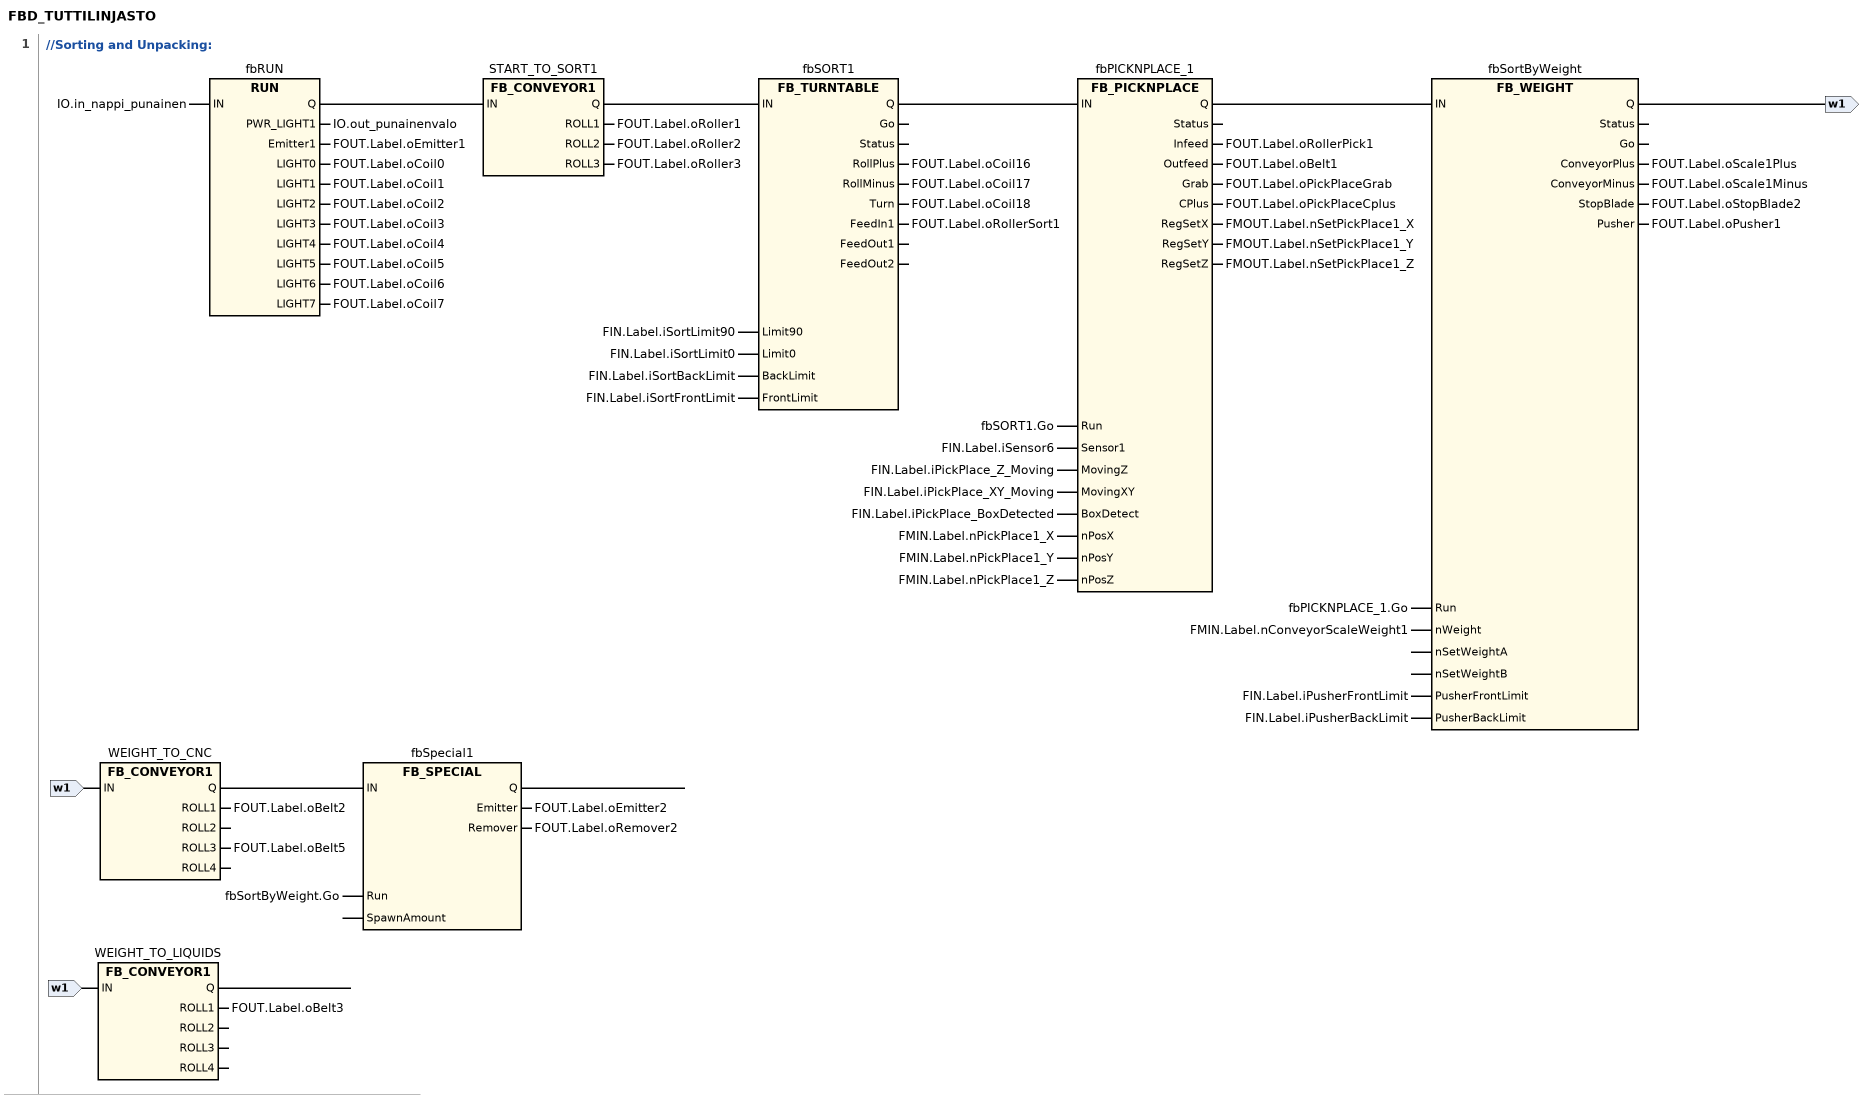
// NETWORK 1
// label: //Sorting and Unpacking
fbRUN(
    IN := IO.in_nappi_punainen,
    PWR_LIGHT1 => IO.out_punainenvalo,
    Emitter1 => FOUT.Label.oEmitter1,
    LIGHT0 => FOUT.Label.oCoil0,
    LIGHT1 => FOUT.Label.oCoil1,
    LIGHT2 => FOUT.Label.oCoil2,
    LIGHT3 => FOUT.Label.oCoil3,
    LIGHT4 => FOUT.Label.oCoil4,
    LIGHT5 => FOUT.Label.oCoil5,
    LIGHT6 => FOUT.Label.oCoil6,
    LIGHT7 => FOUT.Label.oCoil7); // RUN
START_TO_SORT1(
    IN := fbRUN.Q,
    ROLL1 => FOUT.Label.oRoller1,
    ROLL2 => FOUT.Label.oRoller2,
    ROLL3 => FOUT.Label.oRoller3); // FB_CONVEYOR1
fbSORT1(
    IN := START_TO_SORT1.Q,
    Limit90 := FIN.Label.iSortLimit90,
    Limit0 := FIN.Label.iSortLimit0,
    BackLimit := FIN.Label.iSortBackLimit,
    FrontLimit := FIN.Label.iSortFrontLimit,
    RollPlus => FOUT.Label.oCoil16,
    RollMinus => FOUT.Label.oCoil17,
    Turn => FOUT.Label.oCoil18,
    FeedIn1 => FOUT.Label.oRollerSort1); // FB_TURNTABLE
fbPICKNPLACE_1(
    IN := fbSORT1.Q,
    Run := fbSORT1.Go,
    Sensor1 := FIN.Label.iSensor6,
    MovingZ := FIN.Label.iPickPlace_Z_Moving,
    MovingXY := FIN.Label.iPickPlace_XY_Moving,
    BoxDetect := FIN.Label.iPickPlace_BoxDetected,
    nPosX := FMIN.Label.nPickPlace1_X,
    nPosY := FMIN.Label.nPickPlace1_Y,
    nPosZ := FMIN.Label.nPickPlace1_Z,
    Infeed => FOUT.Label.oRollerPick1,
    Outfeed => FOUT.Label.oBelt1,
    Grab => FOUT.Label.oPickPlaceGrab,
    CPlus => FOUT.Label.oPickPlaceCplus,
    RegSetX => FMOUT.Label.nSetPickPlace1_X,
    RegSetY => FMOUT.Label.nSetPickPlace1_Y,
    RegSetZ => FMOUT.Label.nSetPickPlace1_Z); // FB_PICKNPLACE
fbSortByWeight(
    IN := fbPICKNPLACE_1.Q,
    Run := fbPICKNPLACE_1.Go,
    nWeight := FMIN.Label.nConveyorScaleWeight1,
    PusherFrontLimit := FIN.Label.iPusherFrontLimit,
    PusherBackLimit := FIN.Label.iPusherBackLimit,
    ConveyorPlus => FOUT.Label.oScale1Plus,
    ConveyorMinus => FOUT.Label.oScale1Minus,
    StopBlade => FOUT.Label.oStopBlade2,
    Pusher => FOUT.Label.oPusher1); // FB_WEIGHT
WEIGHT_TO_CNC(IN := fbSortByWeight.Q, ROLL1 => FOUT.Label.oBelt2, ROLL3 => FOUT.Label.oBelt5); // FB_CONVEYOR1
fbSpecial1(
    IN := WEIGHT_TO_CNC.Q,
    Run := fbSortByWeight.Go,
    Emitter => FOUT.Label.oEmitter2,
    Remover => FOUT.Label.oRemover2); // FB_SPECIAL
WEIGHT_TO_LIQUIDS(IN := fbSortByWeight.Q, ROLL1 => FOUT.Label.oBelt3); // FB_CONVEYOR1

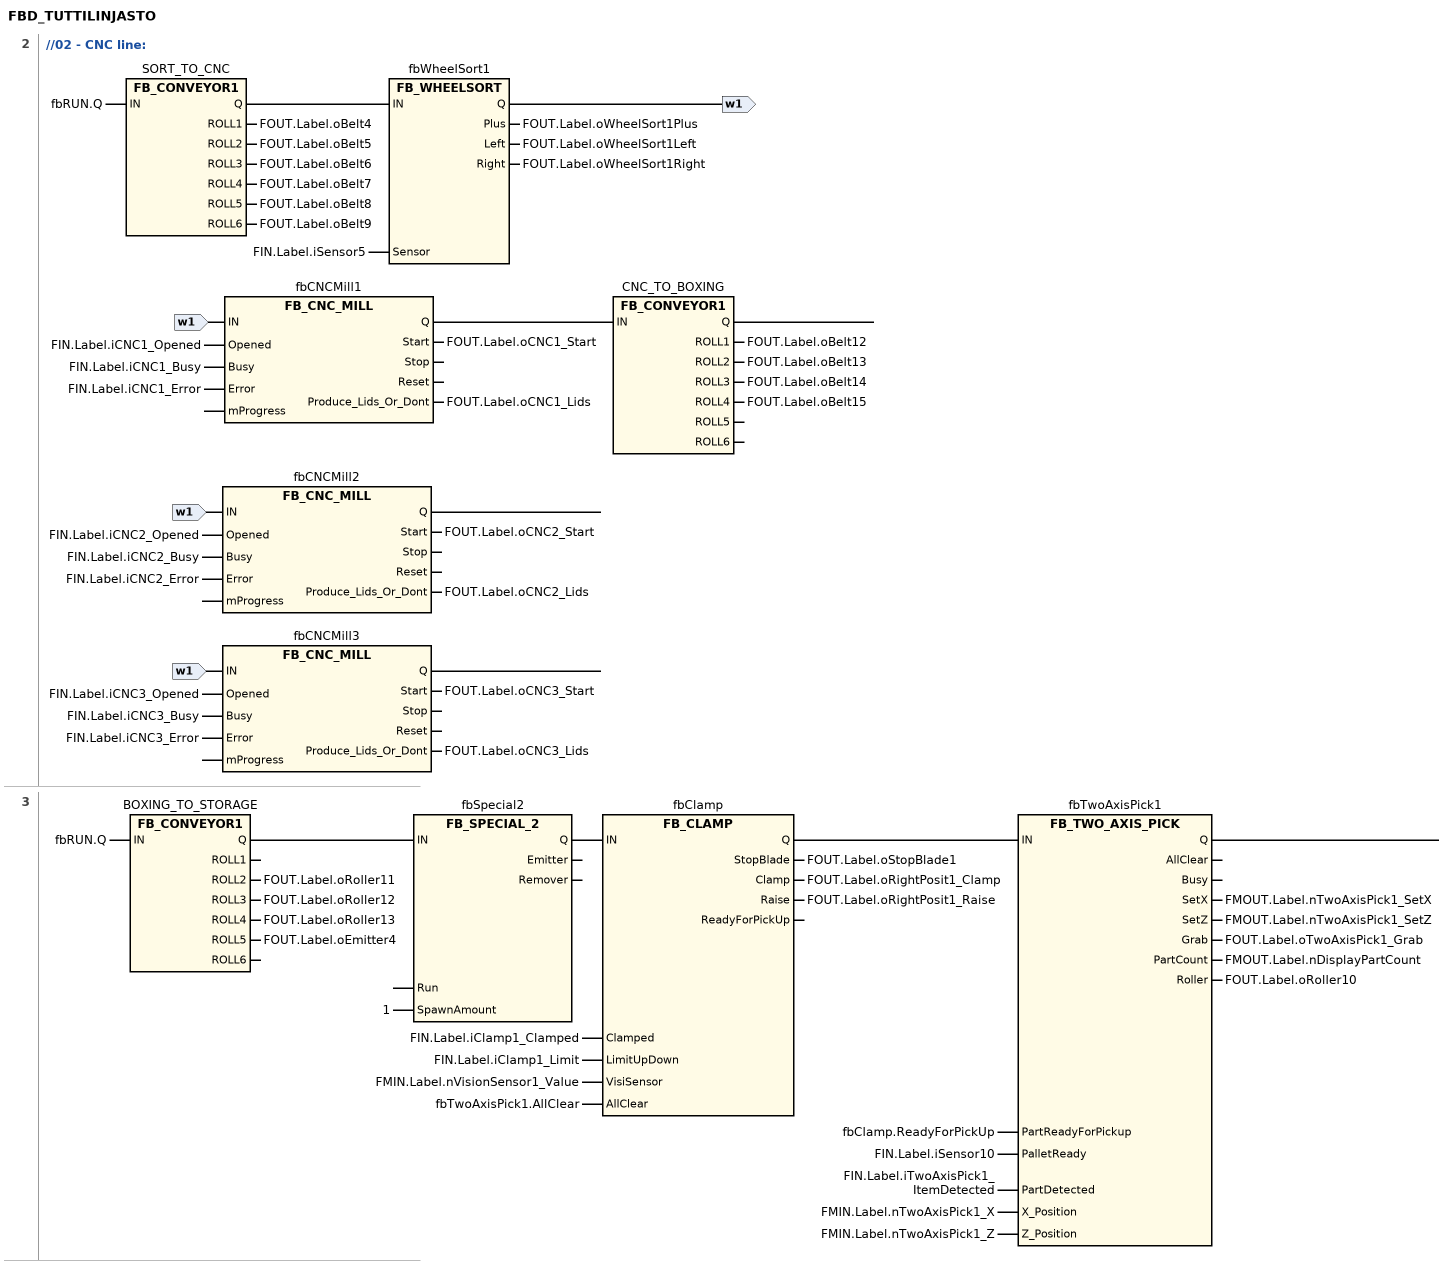
// NETWORK 2
// label: //02 - CNC line
SORT_TO_CNC(
    IN := fbRUN.Q,
    ROLL1 => FOUT.Label.oBelt4,
    ROLL2 => FOUT.Label.oBelt5,
    ROLL3 => FOUT.Label.oBelt6,
    ROLL4 => FOUT.Label.oBelt7,
    ROLL5 => FOUT.Label.oBelt8,
    ROLL6 => FOUT.Label.oBelt9); // FB_CONVEYOR1
fbWheelSort1(
    IN := SORT_TO_CNC.Q,
    Sensor := FIN.Label.iSensor5,
    Plus => FOUT.Label.oWheelSort1Plus,
    Left => FOUT.Label.oWheelSort1Left,
    Right => FOUT.Label.oWheelSort1Right); // FB_WHEELSORT
fbCNCMill1(
    IN := fbWheelSort1.Q,
    Opened := FIN.Label.iCNC1_Opened,
    Busy := FIN.Label.iCNC1_Busy,
    Error := FIN.Label.iCNC1_Error,
    Start => FOUT.Label.oCNC1_Start,
    Produce_Lids_Or_Dont => FOUT.Label.oCNC1_Lids); // FB_CNC_MILL
CNC_TO_BOXING(
    IN := fbCNCMill1.Q,
    ROLL1 => FOUT.Label.oBelt12,
    ROLL2 => FOUT.Label.oBelt13,
    ROLL3 => FOUT.Label.oBelt14,
    ROLL4 => FOUT.Label.oBelt15); // FB_CONVEYOR1
fbCNCMill2(
    IN := fbWheelSort1.Q,
    Opened := FIN.Label.iCNC2_Opened,
    Busy := FIN.Label.iCNC2_Busy,
    Error := FIN.Label.iCNC2_Error,
    Start => FOUT.Label.oCNC2_Start,
    Produce_Lids_Or_Dont => FOUT.Label.oCNC2_Lids); // FB_CNC_MILL
fbCNCMill3(
    IN := fbWheelSort1.Q,
    Opened := FIN.Label.iCNC3_Opened,
    Busy := FIN.Label.iCNC3_Busy,
    Error := FIN.Label.iCNC3_Error,
    Start => FOUT.Label.oCNC3_Start,
    Produce_Lids_Or_Dont => FOUT.Label.oCNC3_Lids); // FB_CNC_MILL

// NETWORK 3
BOXING_TO_STORAGE(
    IN := fbRUN.Q,
    ROLL2 => FOUT.Label.oRoller11,
    ROLL3 => FOUT.Label.oRoller12,
    ROLL4 => FOUT.Label.oRoller13,
    ROLL5 => FOUT.Label.oEmitter4); // FB_CONVEYOR1
fbSpecial2(IN := BOXING_TO_STORAGE.Q, SpawnAmount := 1); // FB_SPECIAL_2
fbClamp(
    IN := fbSpecial2.Q,
    Clamped := FIN.Label.iClamp1_Clamped,
    LimitUpDown := FIN.Label.iClamp1_Limit,
    VisiSensor := FMIN.Label.nVisionSensor1_Value,
    AllClear := fbTwoAxisPick1.AllClear,
    StopBlade => FOUT.Label.oStopBlade1,
    Clamp => FOUT.Label.oRightPosit1_Clamp,
    Raise => FOUT.Label.oRightPosit1_Raise); // FB_CLAMP
fbTwoAxisPick1(
    IN := fbClamp.Q,
    PartReadyForPickup := fbClamp.ReadyForPickUp,
    PalletReady := FIN.Label.iSensor10,
    PartDetected := FIN.Label.iTwoAxisPick1_ItemDetected,
    X_Position := FMIN.Label.nTwoAxisPick1_X,
    Z_Position := FMIN.Label.nTwoAxisPick1_Z,
    SetX => FMOUT.Label.nTwoAxisPick1_SetX,
    SetZ => FMOUT.Label.nTwoAxisPick1_SetZ,
    Grab => FOUT.Label.oTwoAxisPick1_Grab,
    PartCount => FMOUT.Label.nDisplayPartCount,
    Roller => FOUT.Label.oRoller10); // FB_TWO_AXIS_PICK

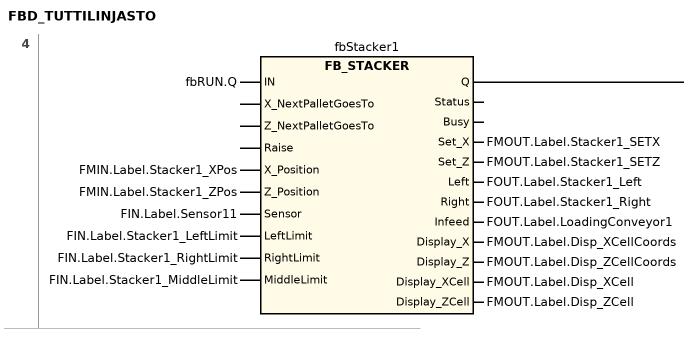
// NETWORK 4
fbStacker1(
    IN := fbRUN.Q,
    X_Position := FMIN.Label.Stacker1_XPos,
    Z_Position := FMIN.Label.Stacker1_ZPos,
    Sensor := FIN.Label.Sensor11,
    LeftLimit := FIN.Label.Stacker1_LeftLimit,
    RightLimit := FIN.Label.Stacker1_RightLimit,
    MiddleLimit := FIN.Label.Stacker1_MiddleLimit,
    Set_X => FMOUT.Label.Stacker1_SETX,
    Set_Z => FMOUT.Label.Stacker1_SETZ,
    Left => FOUT.Label.Stacker1_Left,
    Right => FOUT.Label.Stacker1_Right,
    Infeed => FOUT.Label.LoadingConveyor1,
    Display_X => FMOUT.Label.Disp_XCellCoords,
    Display_Z => FMOUT.Label.Disp_ZCellCoords,
    Display_XCell => FMOUT.Label.Disp_XCell,
    Display_ZCell => FMOUT.Label.Disp_ZCell); // FB_STACKER

END_PROGRAM

// ---- FactoryIO/TUTTITEHDAS/MAIN_TUTTI.TcPOU
PROGRAM MAIN_TUTTI
VAR
	iState: 		INT;	
	iStateName: 	STRING(INT#80);
	iNextState: 	INT;	
//Heartbeats
	iStateHeartBeat: 	DINT;
	TEMP_COUNT: 		DINT;
	ModbusHeartBeat: 	DINT;

//timers
	fbTON1:			TON;
	tStateWait:		TIME := T#0MS;	//TON PT wait duration
	
//Trigs
	rTRIG:			R_TRIG;
	fTRIG:			F_TRIG;
	
	TEMP_TRIG: BOOL;

//Just Modbus Stuff
	ipAddr    : 	STRING(18) := '192.168.0.109';
	bModbusBusy1: 	BOOL;
	bModbusBusy2: 	BOOL;
	bModbusBusy3: 	BOOL;
	bModbusBusy4:	BOOL;
	fbMBReadInputs: 	FB_MBReadInputs;
	fbMBWriteCoils : 	FB_MBWriteCoils;
	fbMBWriteRegs : 	FB_MBWriteRegs;
	fbMBReadInputRegs : FB_MBReadInputRegs;
END_VAR


 CASE iState OF
	0:	//Idle state
	iStateName := 'Idle state';
	iNextState := 10;

	fbTON1(	IN:=TRUE,	PT:= tStateWait);
	IF fbTON1.Q THEN
	fbTON1(IN := FALSE);
		//When timer clicks, do once:
		iStateHeartBeat := iStateHeartBeat+1;
		iState := iNextState;
	END_IF
	
	10:	//READ MODBUS
	iStateName := '10, Read Modbus';
	iNextState := 20;
	fbTON1(	IN:=TRUE,	PT:= tStateWait);
	IF fbTON1.Q THEN
	fbTON1(IN := FALSE);
		//When timer clicks, do once:

		MAIN_TUTTI.MBReadInputs();
		MAIN_TUTTI.MBReadRegisters();
		
		iStateHeartBeat := iStateHeartBeat+1;
		iState := iNextState;
	END_IF
	
	20:	
	iStateName := '20, do stuff more';
	iNextState := 100;
	fbTON1(	IN:=TRUE,	PT:= tStateWait);
	IF fbTON1.Q THEN
	fbTON1(IN := FALSE);
		//When timer clicks, do once:
		
		FBD_TUTTILINJASTO();	//nyt kokeiluna laittaa kaikki roippeet yhteen kivaan pötköön vain, myöhemmin täysin mahdollista pätkiä FBD:t pienempiin osiin
		
		iStateHeartBeat := iStateHeartBeat+1;
		iState := iNextState;
	END_IF		
	
	100: //WRITE MODBUS
	iStateName := '100, Write Modbus';
	iNextState := 0;
	
	fbTON1(	IN:=TRUE,	PT:= tStateWait);
	IF fbTON1.Q THEN
	fbTON1(IN := FALSE);
		//When timer clicks, do once:

		MAIN_TUTTI.MBWriteCoils();
		MAIN_TUTTI.MBWriteRegisters();

		iStateHeartBeat := iStateHeartBeat+1;
		iState := iNextState;
	END_IF

 END_CASE

ACTION MBReadInputs:
IF NOT 	bModbusBusy1 THEN
		bModbusBusy1	:= TRUE;
fbMBReadInputs(
	sIPAddr := ipAddr,
	nTCPPort := 506,
	nUnitID := 255,
	nQuantity := 120,
	nMBAddr := 0,
	cbLength := SIZEOF(TIO.FIN),
	pDestAddr := ADR(TIO.FIN),
	bExecute := TRUE,
	tTimeout := T#1S,
	bBusy => ,
	bError => ,
	nErrId => ,
	cbRead => ,
 );
 ELSE	//jos ModBusBusy ON päällä
	IF NOT fbMBReadInputs.bBusy THEN	//tarkistetaan ettei bBusy ole päällä
		bModbusBusy1	:= FALSE;		//ja mikäli bBusy ei ole päällä niin laitetaan ModbusBusy kans pois
 	END_IF
ModbusHeartBeat := ModbusHeartBeat +1;
fbMBReadInputs(bExecute := FALSE);
END_IF
END_ACTION

ACTION MBReadRegisters:
IF NOT bModbusBusy4 THEN
		bModbusBusy4 				:= TRUE;
fbMBReadInputRegs (
	sIPAddr := ipAddr,
	nTCPPort := 506,
	nUnitID := 255,
	nQuantity := 32,
	nMBAddr := 0,
	cbLength := SIZEOF(TIO.FMIN),
	pDestAddr := ADR(TIO.FMIN),
	bExecute := TRUE,
	tTimeout := T#1S,
	bBusy => ,
	bError => ,
	nErrId => ,
	cbRead => ,
 );
  ELSE
	IF NOT fbMBReadInputRegs.bBusy THEN
		bModbusBusy4	:= FALSE;
 	END_IF
fbMBReadInputRegs(bExecute := FALSE);
END_IF
END_ACTION

ACTION MBWriteCoils:
IF NOT bModbusBusy2 THEN
		bModbusBusy2	:= TRUE;
fbMBWriteCoils(
	sIPAddr := ipAddr,
	nTCPPort := 506,
	nUnitID := 255,
	nQuantity := 120,
	nMBAddr := 0,
	cbLength := SIZEOF(TIO.FOUT),
	pSrcAddr:= ADR(TIO.FOUT), 
	bExecute := TRUE,
	tTimeout := T#1S,
	bBusy=> , 
	bError=> , 
	nErrId=>
);
 ELSE
	IF NOT fbMBWriteCoils.bBusy THEN
		bModbusBusy2	:= FALSE;
 	END_IF
fbMBWriteCoils(bExecute := FALSE);
END_IF
END_ACTION

ACTION MBWriteRegisters:
IF NOT bModbusBusy3 THEN
		bModbusBusy3 				:= TRUE;
fbMBWriteRegs(
	sIPAddr := ipAddr,
	nTCPPort := 506,
	nUnitID := 255,
	nQuantity := 32,
	nMBAddr := 0,
	cbLength := SIZEOF(TIO.FMOUT),
	pSrcAddr:= ADR(TIO.FMOUT), 
	bExecute := TRUE,
	tTimeout := T#1S,
	bBusy=> , 
	bError=> , 
	nErrId=>
);
 ELSE
	IF NOT fbMBWriteRegs.bBusy THEN
		bModbusBusy3				:= FALSE;
 	END_IF
fbMBWriteRegs(bExecute := FALSE);

END_IF


//IF NOT bWriteRegs THEN
// nValue[0]:= nValue[0]+1;
// nValue[1]:= nValue[1]+1;
// nValue[2]:= nValue[2]+1;
// nValue[3]:= nValue[3]+1;

// bWriteRegs :=TRUE;

// fbWriteRegs.sIPAddr :=ipAddr;
// fbWriteRegs.nQuantity := 4;
// fbWriteRegs.nMBAddr := 16#3000;
// fbWriteRegs.cbLength := SIZEOF(nValue);
// fbWriteRegs.pSrcAddr := ADR(nValue);
// fbWriteRegs.tTimeout := T#5s;
// fbWriteRegs(bExecute:=TRUE);
//ELSE
// IF NOT fbWriteRegs.bBUSY THEN
// bWriteRegs :=FALSE;
//END_IF
// fbWriteRegs(bExecute:=FALSE);
//END_IF
END_ACTION

ACTION WAIT:
//ACTION WAIT
//Poistetaan testi-Action pois käytöstä.
//On parempi pääkoodissa näkyä mitä tapahtuu, ja tämä funktio selkeästi muuttuu jatkuvasti

//fbTON1(	IN:=TRUE,
//		PT:= tWaitTime);
//	IF fbTON1.Q THEN
//		fbTON1(IN := FALSE);
//		iStateCounter := iStateCounter+1;
//		iState := iNextState;
//	END_IF
END_ACTION

END_PROGRAM
